(* CoDeSys 2.3.9.28 project: MagsaSTPRO.pro *)
(* Libraries: SysLibTime.lib 27.1.09 09:27:38, Iecsfc.lib 24.11.08 06:07:15, Festo_Motion.lib 17.8.11 07:30:49, 3S_CANopenMaster.lib 3.4.14 07:23:31, 3S_CANopenManager.lib 3.12.10 12:40:14, Standard.lib 27.1.09 09:27:38, Util.lib 27.1.09 09:27:38, SysTaskInfo.lib 24.11.08 06:07:15, SYSLIBCALLBACK.LIB 27.1.09 09:27:38, 3S_CanDrv.lib 3.7.09 09:28:00 *)

(* PLC configuration (modules and I/O channels)
Hexswitch AT %IB0 [HexSwitch] rotary switch 0 = STOP, 1-15 = RUN
AT %IB4 [ByteInput] -
AT %QB0 [ByteOutput] -
AT %IB8 [ByteInput] -
AT %QB4 [ByteOutput] -
*)

(* Task configuration *)
TASK NewTask (PRIORITY := 10, INTERVAL := T#8ms);
	bombas();
	Podium();
	PLC_PRG();
END_TASK

(* Global variable list: CanOpen implicit Variables *)
VAR_GLOBAL CONSTANT
	MAX_CTRLINDEX : INT := 0;
END_VAR
VAR_GLOBAL CONSTANT
	USE_CANOPEN_NODES : BOOL := TRUE;
	MAX_MASTERINDEX : INT := 0;
	MAX_NODEINDEX : INT := 1;
	MAX_SDOINDEX : INT := 37;
	MAX_PDOINDEX_RX : INT := 7;
	MAX_PDOINDEX_TX : INT := 7;
	MAX_MASTER_ODENTRY_IDX : INT := 0;
END_VAR
VAR_GLOBAL
	pCANopenMaster : ARRAY[0..MAX_MASTERINDEX] OF CanOpenMaster;
	pCanOpenNode : ARRAY[0..MAX_NODEINDEX] OF CanOpenNode;
	pCanOpenSDO : ARRAY[0..MAX_SDOINDEX] OF CanOpenSDO;
	pCanOpenPDO_Rx : ARRAY[0..MAX_PDOINDEX_RX] OF CanOpenPDO_Rx;
	pCanOpenPDO_Tx : ARRAY[0..MAX_PDOINDEX_TX] OF CanOpenPDO_Tx;
	 ODMEntries: ARRAY[0..MAX_MASTER_ODENTRY_IDX] OF CanOpenODEntry;
END_VAR

(* Global variable list: Global_Variables *)
VAR_GLOBAL

	EjecutaM1_Pos1: BOOL;
	EjecutaM1_Pos2: BOOL;
	EjecutaM1_Pos3: BOOL;
	EjecutaM1_Pos4: BOOL;
	EjecutaM1_Pos5: BOOL;
	EjecutaM1_Pos6: BOOL;
	EjecutaM1_Pos7: BOOL;
	EjecutaM1_Pos8: BOOL;
	EjecutaM1_Pos9: BOOL;
	EjecutaM1_Pos10: BOOL;



	EjecutaM2_Pos1: BOOL;
	EjecutaM2_Pos2: BOOL;
	EjecutaM2_Pos3: BOOL;
	EjecutaM2_Pos4: BOOL;
	EjecutaM2_Pos5: BOOL;
	EjecutaM2_Pos6: BOOL;
	EjecutaM2_Pos7: BOOL;
	EjecutaM2_Pos8: BOOL;
	EjecutaM2_Pos9: BOOL;
	EjecutaM2_Pos10: BOOL;

	SecuenciaMotor1: INT;
	SecuenciaMotor2: INT;



END_VAR


VAR_GLOBAL RETAIN PERSISTENT

	HMI_M1_POS_1: DINT;
	HMI_M1_POS_2: DINT;
	HMI_M1_POS_3: DINT;
	HMI_M1_POS_4: DINT;
	HMI_M1_POS_5: DINT;
	HMI_M1_POS_6: DINT;
	HMI_M1_POS_7: DINT;
	HMI_M1_POS_8: DINT;
	HMI_M1_POS_9: DINT;
	HMI_M1_POS_10: DINT;

	HMI_M1_VEL_1: USINT;
	HMI_M1_VEL_2: USINT;
	HMI_M1_VEL_3: USINT;
	HMI_M1_VEL_4: USINT;
	HMI_M1_VEL_5: USINT;
	HMI_M1_VEL_6: USINT;
	HMI_M1_VEL_7: USINT;
	HMI_M1_VEL_8: USINT;
	HMI_M1_VEL_9: USINT;
	HMI_M1_VEL_10: USINT;

	HMI_M2_POS_1: DINT;
	HMI_M2_POS_2: DINT;
	HMI_M2_POS_3: DINT;
	HMI_M2_POS_4: DINT;
	HMI_M2_POS_5: DINT;
	HMI_M2_POS_6: DINT;
	HMI_M2_POS_7: DINT;
	HMI_M2_POS_8: DINT;
	HMI_M2_POS_9: DINT;
	HMI_M2_POS_10: DINT;

	HMI_M2_VEL_1: USINT;
	HMI_M2_VEL_2: USINT;
	HMI_M2_VEL_3: USINT;
	HMI_M2_VEL_4: USINT;
	HMI_M2_VEL_5: USINT;
	HMI_M2_VEL_6: USINT;
	HMI_M2_VEL_7: USINT;
	HMI_M2_VEL_8: USINT;
	HMI_M2_VEL_9: USINT;
	HMI_M2_VEL_10: USINT;

	Stop: BOOL;


END_VAR

(* POU bombas, ST *)
PROGRAM bombas
VAR
	HMI_ColorRojo: BOOL;
	In_Rojo AT %IX2.1: BOOL;
	HMI_ColorAzul: BOOL;
	In_Azul AT %IX2.2: BOOL;
	HMI_ColorAmarillo: BOOL;
	In_Amarillo AT %IX2.3: BOOL;
	EmpezarJuego: BOOL;
	Explota AT %QX0.1: BOOL;
	juego: INT;
	tiempoBomba1: TON;
	tiempoBomba2: TON;
END_VAR
IF NOT EmpezarJuego THEN
juego:=0;
tiempoBomba1(in:=FALSE, pt:=t#0s);
tiempoBomba2(in:=FALSE, pt:=t#0s);
Explota:=FALSE;
END_IF


CASE juego OF

0:

IF In_rojo AND In_azul AND In_amarillo AND EmpezarJuego THEN
tiempoBomba1(in:=FALSE, pt:=t#0s);
tiempoBomba2(in:=FALSE, pt:=t#0s);
Explota:=FALSE;
juego:=11;
END_IF


11:
IF HMI_ColorRojo AND NOT In_Rojo AND EmpezarJuego THEN
juego:=1;
END_IF

IF HMI_ColorAzul AND NOT In_Azul AND EmpezarJuego THEN
juego:=1;
END_IF

IF HMI_ColorAmarillo AND NOT In_Amarillo AND EmpezarJuego THEN
juego:=1;
END_IF

1:
tiempoBomba1(in:=TRUE, pt:=t#1s);
IF tiempoBomba1.Q THEN
Explota:=TRUE;
tiempoBomba1(in:=FALSE, pt:=t#0s);
juego:=2;
END_IF

2:
tiempoBomba2(in:=TRUE, pt:=t#4s);
IF tiempoBomba2.Q THEN
Explota:=FALSE;
tiempoBomba2(in:=FALSE, pt:=t#0s);
juego:=0;
END_IF

END_CASE
END_PROGRAM

(* POU Podium, ST *)
PROGRAM Podium
VAR

	ActivarMecanismo: BOOL;

	subePodium: BOOL;
	bajaPodium: BOOL;

	tiempo1: TON;
	tiempo2: TON;
	tiempo3: TON;
	tiempo4: TON;
	tiempo5: TON;


	bobina1 AT %QX0.0: BOOL;
	bobina2 AT %QX0.2: BOOL;

	sube: INT;
	baja: INT;

	abre: INT;
	cierra: INT;
	forzarAbrir: BOOL;
	forzarCerrar: BOOL;
END_VAR
IF NOT ActivarMecanismo THEN

	tiempo1(in:=FALSE, pt:=t#0s);
	tiempo2(in:=FALSE, pt:=t#0s);
	tiempo3(in:=FALSE, pt:=t#0s);
	tiempo4(in:=FALSE, pt:=t#0s);
	bobina1:=FALSE;
	bobina2:=FALSE;
	subePodium:= FALSE;
	bajaPodium:= FALSE;


END_IF


CASE abre OF

	0:
	IF forzarAbrir THEN
		abre:=1;
	END_IF

	1:
	tiempo1(in:=TRUE, pt:=t#1s);
	IF tiempo1.Q THEN
		bobina1:=TRUE;
		tiempo1(in:=FALSE, pt:=t#0s);
		abre:=2;
	END_IF

	2:
	tiempo2(in:=TRUE, pt:=t#2s);
	IF tiempo2.Q THEN
		bobina2:=TRUE;
		tiempo2(in:=FALSE, pt:=t#0s);
		forzarAbrir:= FALSE;
		abre:=0;
	END_IF

END_CASE

CASE cierra OF
	0:
	IF forzarCerrar THEN
		cierra:=1;
	END_IF

	1:
	tiempo3(in:=TRUE, pt:=t#1s);
	IF tiempo3.Q THEN
		bobina2:=FALSE;
		tiempo3(in:=FALSE, pt:=t#0s);
		cierra:=2;
	END_IF


	2:
	tiempo4(in:=TRUE, pt:=t#3s);
	IF tiempo4.Q THEN
		bobina1:=FALSE;
		tiempo4(in:=FALSE, pt:=t#0s);
		cierra:=0;
		forzarCerrar:= FALSE;
	END_IF

END_CASE


CASE sube OF

	0:
	IF ActivarMecanismo AND  subePodium AND NOT bajaPodium THEN
		sube:=1;
	END_IF

	1:
	forzarAbrir:= TRUE;
	tiempo3(in:=TRUE, pt:=t#1s);
	IF abre = 0 THEN
		tiempo3(in:=FALSE, pt:=t#0s);
		sube:=2;
	END_IF

	2:
	tiempo4(in:=TRUE, pt:=t#4s);
	IF tiempo4.Q THEN
		EjecutaM2_Pos1:= TRUE;
		tiempo4(in:=FALSE, pt:=t#0s);
		sube:=3;
	END_IF

	3:
	tiempo5(in:=TRUE, pt:=t#1s);
	IF tiempo5.Q THEN
		EjecutaM2_Pos1:= FALSE;
		tiempo5(in:=FALSE, pt:=t#0s);
		sube:=4;
	END_IF

	4:
	subePodium:=FALSE;
	sube:= 0;

END_CASE


CASE baja OF

	0:

	IF ActivarMecanismo AND bajaPodium AND NOT subePodium THEN
		baja:=1;
	END_IF


	1:
	tiempo1(in:=TRUE, pt:=t#1s);
	IF tiempo1.Q THEN
		EjecutaM2_Pos2:= TRUE;
		tiempo1(in:=FALSE, pt:=t#0s);
		baja:=2;
	END_IF

	2:
	tiempo2(in:=TRUE, pt:=t#2s);
	IF tiempo2.Q AND SecuenciaMotor2 = 0 THEN
		EjecutaM2_Pos2:= FALSE;
		tiempo2(in:=FALSE, pt:=t#0s);
		baja:=3;
	END_IF

	3:
	forzarCerrar:= TRUE;
	tiempo5(in:=TRUE, pt:=t#1s);
	IF cierra = 0 THEN
		tiempo5(in:=FALSE, pt:=t#0s);
		baja:=4;
	END_IF

	4:
	bajaPodium:=FALSE;
	baja:= 0;

END_CASE
END_PROGRAM

(* POU PLC_PRG, ST *)
PROGRAM PLC_PRG
VAR


	Motor1: CMMP_AS_CTRL;
	Motor2: CMMP_AS_CTRL;
	Out1 AT %QB8: BYTE;
	In1 AT %IB12: BYTE;
	Out2 AT %QB40: BYTE;
	In2 AT %IB44: BYTE;

	(* HMI *)

	HMI_ParoEmergencia: BOOL;
	HMI_Habilitar1: BOOL;
	HMI_Habilitar2: BOOL;
	HMI_JoggPos1: BOOL;
	HMI_JoggNeg1: BOOL;
	HMI_JoggPos2: BOOL;
	HMI_JoggNeg2: BOOL;
	HMI_Home1: BOOL;
	HMI_Home2: BOOL;

	Falla1: BOOL;
	Falla2: BOOL;
	Listo1: BOOL;
	Listo2: BOOL;
	Reset1: BOOL;
	Reset2: BOOL;
	Habilitado1: BOOL;
	Habilitado2: BOOL;
	Referenciado1: BOOL;
	Referenciado2: BOOL;

	PosicionActual1: DINT;
	PosicionActual2: DINT;
	VelocidadActual1: SINT;
	VelocidadActual2: SINT;


	timeEspera1: TON;
	timeEspera2: TON;

END_VAR
(* INIT *)
Motor1(FHPP_In:=In1, FHPP_Out:=Out1);
Motor2(FHPP_In:=In2, FHPP_Out:=Out2);

(* D R I V E R S *)

(* MOTOR 1 *)


Motor1.Halt := HMI_Habilitar1;
Motor1.EnableDrive:=HMI_Habilitar1;
Motor1.Stop:=HMI_Habilitar1;
Motor1.ResetFault := reset1;
Motor1.OPM := 1;
Motor1.AbsoluteRelative := 0;
Habilitado1:= Motor1.DriveEnabled;
Listo1:= Motor1.Ready;
Falla1:= Motor1.Fault;
Referenciado1:= Motor1.DriveIsReferenced;
PosicionActual1:= Motor1.ActualPosition;
VelocidadActual1:= Motor1.ActualVelocity;


(* MOTOR 2 *)

Motor2.EnableDrive := HMI_Habilitar2;
Motor2.Halt := HMI_Habilitar2;
Motor2.Stop:=HMI_Habilitar2;
Motor2.ResetFault := reset2;
Motor2.OPM := 1;
Motor2.AbsoluteRelative := 0;
Habilitado2:= Motor2.DriveEnabled;
Listo2:= Motor2.Ready;
Falla2:= Motor2.Fault;
Referenciado2:= Motor2.DriveIsReferenced;
PosicionActual2:= Motor2.ActualPosition;
VelocidadActual2:= Motor2.ActualVelocity;


IF stop THEN
	Motor1.EnableDrive:=FALSE;
	Motor1.Stop:=FALSE;
	Motor1.Halt:=FALSE;
	Motor2.EnableDrive:=FALSE;
	Motor2.Stop:=FALSE;
	Motor2.Halt:=FALSE;
	HMI_Habilitar1:=FALSE;
	HMI_Habilitar2:=FALSE;
	SecuenciaMotor1:=0;
	SecuenciaMotor2:=0;
END_IF

IF NOT stop THEN
	HMI_Habilitar1:=TRUE;
	HMI_Habilitar2:=TRUE;
END_IF


(*jogg positivo 1*)
IF HMI_JoggPos1 AND Motor1.Ready THEN
	motor1.JoggingPos:=TRUE;
ELSE
	motor1.JoggingPos:=FALSE;
END_IF
(*jogg negativo 1*)
IF HMI_JoggNeg1 AND Motor1.Ready THEN
	motor1.JoggingNeg:=TRUE;
ELSE
	motor1.JoggingNeg:=FALSE;
END_IF

(*jogg positivo 2*)
IF HMI_JoggPos2 AND Motor2.Ready THEN
	motor2.JoggingPos:=TRUE;
ELSE
	motor2.JoggingPos:=FALSE;
END_IF
(*jogg negativo 2*)
IF HMI_JoggNeg2 AND Motor2.Ready THEN
	motor2.JoggingNeg:=TRUE;
ELSE
	motor2.JoggingNeg:=FALSE;
END_IF
(*home 1*)
IF HMI_Home1 AND Motor1.Ready THEN
	motor1.StartHoming:=TRUE;
ELSE
	motor1.StartHoming:=FALSE;
END_IF
(*home 2*)
IF HMI_Home2 AND Motor2.Ready THEN
	motor2.StartHoming:=TRUE;
ELSE
motor2.StartHoming:=FALSE;
END_IF


CASE SecuenciaMotor1 OF

	0:
	IF EjecutaM1_Pos1 AND habilitado1 AND listo1 AND NOT falla1 THEN
		Motor1.SetValuePosition:=HMI_M1_POS_1;
		Motor1.SetValueVelocity:=HMI_M1_VEL_1;
		Motor1.StartTask:=FALSE;
		SecuenciaMotor1:=1;
	END_IF

	IF EjecutaM1_Pos2 AND habilitado1 AND listo1 AND NOT falla1 THEN
		motor1.SetValuePosition:=HMI_M1_POS_2;
		motor1.SetValueVelocity:=HMI_M1_VEL_2;
		motor1.StartTask:=FALSE;
		SecuenciaMotor1:=1;
	END_IF

	IF EjecutaM1_Pos3 AND habilitado1 AND listo1 AND NOT falla1 THEN
		motor1.SetValuePosition:=HMI_M1_POS_3;
		motor1.SetValueVelocity:=HMI_M1_VEL_3;
		motor1.StartTask:=FALSE;
		SecuenciaMotor1:=1;
	END_IF


	IF EjecutaM1_Pos4 AND habilitado1 AND listo1 AND NOT falla1 THEN
		motor1.SetValuePosition:=HMI_M1_POS_4;
		motor1.SetValueVelocity:=HMI_M1_VEL_4;
		motor1.StartTask:=FALSE;
		SecuenciaMotor1:=1;
	END_IF


	IF EjecutaM1_Pos5 AND habilitado1 AND listo1 AND NOT falla1 THEN
		motor1.SetValuePosition:=HMI_M1_POS_5;
		motor1.SetValueVelocity:=HMI_M1_VEL_5;
		motor1.StartTask:=FALSE;
		SecuenciaMotor1:=1;
	END_IF


	IF EjecutaM1_Pos6 AND habilitado1 AND listo1 AND NOT falla1 THEN
		motor1.SetValuePosition:=HMI_M1_POS_6;
		motor1.SetValueVelocity:=HMI_M1_VEL_6;
		motor1.StartTask:=FALSE;
		SecuenciaMotor1:=1;
	END_IF


	IF EjecutaM1_Pos7 AND habilitado1 AND listo1 AND NOT falla1 THEN
		motor1.SetValuePosition:=HMI_M1_POS_7;
		motor1.SetValueVelocity:=HMI_M1_VEL_7;
		motor1.StartTask:=FALSE;
		SecuenciaMotor1:=1;
	END_IF


	IF EjecutaM1_Pos8 AND habilitado1 AND listo1 AND NOT falla1 THEN
		motor1.SetValuePosition:=HMI_M1_POS_8;
		motor1.SetValueVelocity:=HMI_M1_VEL_8;
		motor1.StartTask:=FALSE;
		SecuenciaMotor1:=1;
	END_IF

	IF EjecutaM1_Pos9 AND habilitado1 AND listo1 AND NOT falla1 THEN
		motor1.SetValuePosition:=HMI_M1_POS_9;
		motor1.SetValueVelocity:=HMI_M1_VEL_9;
		motor1.StartTask:=FALSE;
		SecuenciaMotor1:=1;
	END_IF

	IF EjecutaM1_Pos10 AND habilitado1 AND listo1 AND NOT falla1 THEN
		motor1.SetValuePosition:=HMI_M1_POS_10;
		motor1.SetValueVelocity:=HMI_M1_VEL_10;
		motor1.StartTask:=FALSE;
		SecuenciaMotor1:=1;
	END_IF


	1:
	IF NOT motor1.DriveIsMoving THEN
		timeEspera1(in:=FALSE, pt:=t#0s);
		SecuenciaMotor1:=2;
	END_IF

	2:
	timeEspera1(in:=TRUE, pt:=t#100ms);
	IF timeEspera1.Q AND motor1.MC THEN
		timeEspera1(in:=FALSE, pt:=t#0s);
		motor1.StartTask:=TRUE;
		SecuenciaMotor1:=3;
	END_IF

	3:
	IF motor1.MC AND NOT  motor1.DriveIsMoving THEN
		motor1.StartTask:=FALSE;
		SecuenciaMotor1:=0;
	END_IF

END_CASE


CASE SecuenciaMotor2 OF

	0:
	IF EjecutaM2_Pos1 AND habilitado2 AND listo2 AND NOT falla2 THEN
		Motor2.SetValuePosition:=HMI_M2_POS_1;
		Motor2.SetValueVelocity:=HMI_M2_VEL_1;
		Motor2.StartTask:=FALSE;
		SecuenciaMotor2:=1;
	END_IF

	IF EjecutaM2_Pos2 AND habilitado2 AND listo2 AND NOT falla2 THEN
		motor2.SetValuePosition:=HMI_M2_POS_2;
		motor2.SetValueVelocity:=HMI_M2_VEL_2;
		motor2.StartTask:=FALSE;
		SecuenciaMotor2:=1;
	END_IF

	IF EjecutaM2_Pos3 AND habilitado2 AND listo2 AND NOT falla2 THEN
		motor2.SetValuePosition:=HMI_M2_POS_3;
		motor2.SetValueVelocity:=HMI_M2_VEL_3;
		motor2.StartTask:=FALSE;
		SecuenciaMotor2:=1;
	END_IF




	IF EjecutaM2_Pos4 AND habilitado2 AND listo2 AND NOT falla2 THEN
		motor2.SetValuePosition:=HMI_M2_POS_4;
		motor2.SetValueVelocity:=HMI_M2_VEL_4;
		motor2.StartTask:=FALSE;
		SecuenciaMotor2:=1;
	END_IF


	IF EjecutaM2_Pos5 AND habilitado2 AND listo2 AND NOT falla2 THEN
		motor2.SetValuePosition:=HMI_M2_POS_5;
		motor2.SetValueVelocity:=HMI_M2_VEL_5;
		motor2.StartTask:=FALSE;
		SecuenciaMotor2:=1;
	END_IF


	IF EjecutaM2_Pos6 AND habilitado2 AND listo2 AND NOT falla2 THEN
		motor2.SetValuePosition:=HMI_M2_POS_6;
		motor2.SetValueVelocity:=HMI_M2_VEL_6;
		motor2.StartTask:=FALSE;
		SecuenciaMotor2:=1;
	END_IF



	IF EjecutaM2_Pos7 AND habilitado2 AND listo2 AND NOT falla2 THEN
		motor2.SetValuePosition:=HMI_M2_POS_7;
		motor2.SetValueVelocity:=HMI_M2_VEL_7;
		motor2.StartTask:=FALSE;
		SecuenciaMotor2:=1;
	END_IF


	IF EjecutaM2_Pos8 AND habilitado2 AND listo2 AND NOT falla2 THEN
		motor2.SetValuePosition:=HMI_M2_POS_8;
		motor2.SetValueVelocity:=HMI_M2_VEL_8;
		motor2.StartTask:=FALSE;
		SecuenciaMotor2:=1;
	END_IF

	IF EjecutaM2_Pos9 AND habilitado2 AND listo2 AND NOT falla2 THEN
		motor2.SetValuePosition:=HMI_M2_POS_9;
		motor2.SetValueVelocity:=HMI_M2_VEL_9;
		motor2.StartTask:=FALSE;
		SecuenciaMotor2:=1;
	END_IF

	IF EjecutaM2_Pos10 AND habilitado2 AND listo2 AND NOT falla2 THEN
		motor2.SetValuePosition:=HMI_M2_POS_10;
		motor2.SetValueVelocity:=HMI_M2_VEL_10;
		motor2.StartTask:=FALSE;
		SecuenciaMotor2:=1;
	END_IF


	1:
	IF NOT motor2.DriveIsMoving THEN
		timeEspera2(in:=FALSE, pt:=t#0s);
		SecuenciaMotor2:=2;
	END_IF

	2:
	timeEspera2(in:=TRUE, pt:=t#100ms);
	IF timeEspera2.Q AND motor2.MC THEN
		timeEspera2(in:=FALSE, pt:=t#0s);
		motor2.StartTask:=TRUE;
		SecuenciaMotor2:=3;
	END_IF

	3:
	IF motor2.MC AND NOT  motor2.DriveIsMoving THEN
		motor2.StartTask:=FALSE;
		SecuenciaMotor2:=0;
	END_IF

END_CASE
END_PROGRAM
